FUNCTION_BLOCK INTERNAL FB_SFC_PressDemoAuto EXTENDS FB_SequenceBase
VAR_INPUT
END_VAR
VAR_OUTPUT
END_VAR
VAR
END_VAR

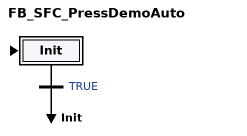
INITIAL_STEP Init:
END_STEP
TRANSITION FROM Init TO Init
    := TRUE;
END_TRANSITION

END_FUNCTION_BLOCK

(* stored: Version 1.1.0.1
   POU FB_SFC_PressDemoAuto: Id {5a6ce38f-33a5-4b54-b6a4-05132bef8883}, SpecialFunc None *)
